TYPE ST_LaudaWriteCommands_Control :
STRUCT
	SetpointOffset	: STRING := 'OUT_PAR_14_';
	ControlVariable	: STRING := 'OUT_MODE_01_X';
	OffsetSource	: string := 'OUT_MODE_04_X';
END_STRUCT
END_TYPE

(* stored: Version 1.1.0.1, ProductVersion 3.1.4024.12
   DUT ST_LaudaWriteCommands_Control: Id {6d00b474-04b1-440f-baf7-e79bbcb04843} *)
